TYPE structEventViewMsg :
STRUCT
	//combined implementation
	msgArry: ARRAY[1..gHMIData.gNumberOfMessagesScreen] OF typeNewMsg;
	msgArryStyle: ARRAY[1..gHMIData.gNumberOfMessagesScreen] OF typeNewMsgStyle;
	msgHeader:typeNewMsgHeader;
END_STRUCT
END_TYPE

(* stored: Version 1.1.0.1, ProductVersion 3.1.4024.12
   DUT structEventViewMsg: Id {ed70df21-0d48-484e-85f3-d55ac78a9628} *)
